// TIA Portal V15.1 export
// export: Created 2020-06-12T07:35:51.5537109Z, ExportSetting None, DisplayName Totally Integrated Automation Portal, DisplayVersion V15.1, DisplayName TIA Portal Openness, DisplayVersion V15.1, DisplayName STEP 7 Professional, DisplayVersion V15.1, DisplayName STEP 7 Safety, DisplayVersion V15.1, DisplayName WinCC Advanced, DisplayVersion V15.1
FUNCTION "MELT_Locks" : Void   // FC50, FBD
{ S7_Optimized_Access := 'TRUE' }
// stored: SetENOAutomatically False
   VAR_TEMP
      tCBisDisabled : Bool;
      tCBisLocked : Bool;
      tCWTripByMS : Bool;
      tCWPumpsStop : Bool;
      tMeltTripReset : Bool;
      tMpStatus : Word;
      tMeltTrip : Bool;
      tReset : Bool;
      tLC5MeltMode : Bool;
      tMSNotUsed : Bool;
   END_VAR
BEGIN

REGION Network 1: Reset trips
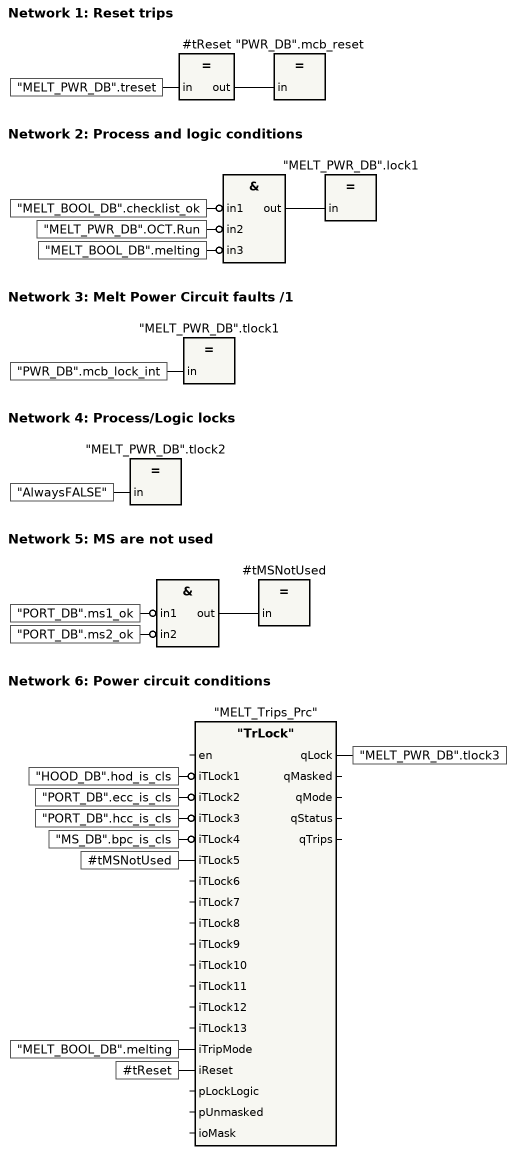
   #tReset := "MELT_PWR_DB".treset;
   "PWR_DB".mcb_reset := "MELT_PWR_DB".treset;
END_REGION

REGION Network 2: Process and logic conditions
   "MELT_PWR_DB".lock1 := NOT "MELT_BOOL_DB".checklist_ok AND NOT "MELT_PWR_DB".OCT.Run AND NOT "MELT_BOOL_DB".melting;
END_REGION

REGION Network 3: Melt Power Circuit faults /1
   "MELT_PWR_DB".tlock1 := "PWR_DB".mcb_lock_int;
END_REGION

REGION Network 4: Process/Logic locks
   // THIS IS TEMPORARY
   "MELT_PWR_DB".tlock2 := "AlwaysFALSE";
END_REGION

REGION Network 5: MS are not used
   #tMSNotUsed := NOT "PORT_DB".ms1_ok AND NOT "PORT_DB".ms2_ok;
END_REGION

REGION Network 6: Power circuit conditions
   "MELT_Trips_Prc"(iTLock1 := NOT "HOOD_DB".hod_is_cls,   // "TrLock"
                    iTLock2 := NOT "PORT_DB".ecc_is_cls,
                    iTLock3 := NOT "PORT_DB".hcc_is_cls,
                    iTLock4 := NOT "MS_DB".bpc_is_cls,
                    iTLock5 := #tMSNotUsed,
                    iTripMode := "MELT_BOOL_DB".melting,
                    iReset := #tReset,
                    qLock => "MELT_PWR_DB".tlock3);
END_REGION

REGION Network 7: Cooling common trips
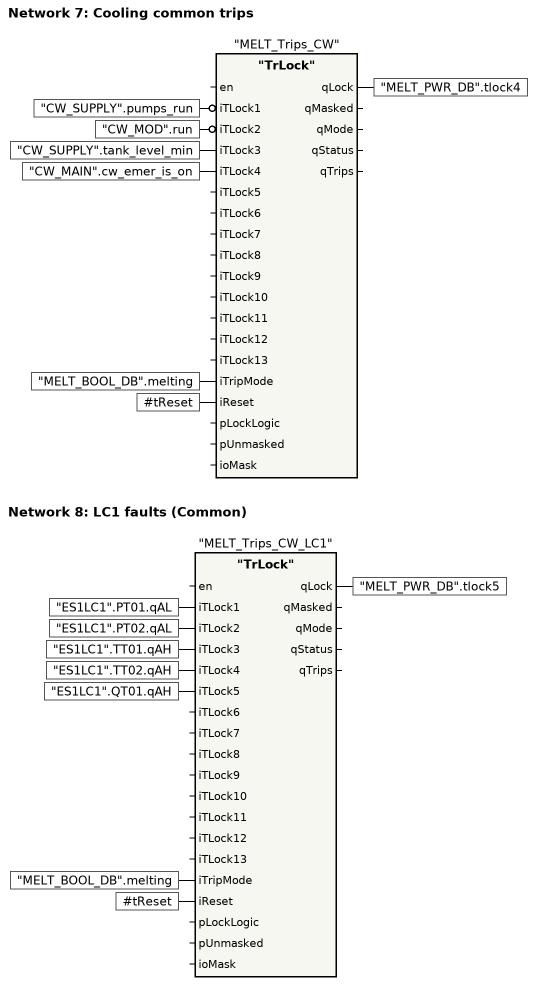
   "MELT_Trips_CW"(iTLock1 := NOT "CW_SUPPLY".pumps_run,   // "TrLock"
                   iTLock2 := NOT "CW_MOD".run,
                   iTLock3 := "CW_SUPPLY".tank_level_min,
                   iTLock4 := "CW_MAIN".cw_emer_is_on,
                   iTripMode := "MELT_BOOL_DB".melting,
                   iReset := #tReset,
                   qLock => "MELT_PWR_DB".tlock4);
END_REGION

REGION Network 8: LC1 faults (Common)
   // "ES1LC1".TT03.qAH
   // "ES1LC1".TT04.qAH
   "MELT_Trips_CW_LC1"(iTLock1 := "ES1LC1".PT01.qAL,   // "TrLock"
                       iTLock2 := "ES1LC1".PT02.qAL,
                       iTLock3 := "ES1LC1".TT01.qAH,
                       iTLock4 := "ES1LC1".TT02.qAH,
                       iTLock5 := "ES1LC1".QT01.qAH,
                       iTripMode := "MELT_BOOL_DB".melting,
                       iReset := #tReset,
                       qLock => "MELT_PWR_DB".tlock5);
END_REGION

REGION Network 9: LC3 faults (Portal + HC-clamps)
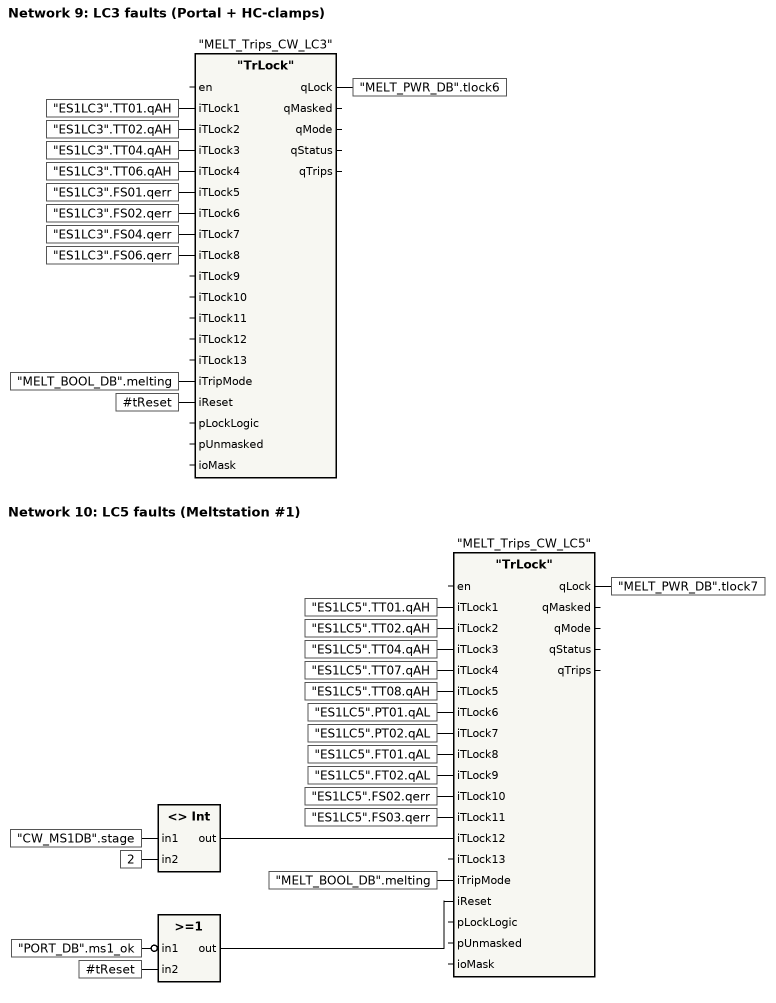
   "MELT_Trips_CW_LC3"(iTLock1 := "ES1LC3".TT01.qAH,   // "TrLock"
                       iTLock2 := "ES1LC3".TT02.qAH,
                       iTLock3 := "ES1LC3".TT04.qAH,
                       iTLock4 := "ES1LC3".TT06.qAH,
                       iTLock5 := "ES1LC3".FS01.qerr,
                       iTLock6 := "ES1LC3".FS02.qerr,
                       iTLock7 := "ES1LC3".FS04.qerr,
                       iTLock8 := "ES1LC3".FS06.qerr,
                       iTripMode := "MELT_BOOL_DB".melting,
                       iReset := #tReset,
                       qLock => "MELT_PWR_DB".tlock6);
END_REGION

REGION Network 10: LC5 faults (Meltstation #1)
   "MELT_Trips_CW_LC5"(iTLock1 := "ES1LC5".TT01.qAH,   // "TrLock"
                       iTLock2 := "ES1LC5".TT02.qAH,
                       iTLock3 := "ES1LC5".TT04.qAH,
                       iTLock4 := "ES1LC5".TT07.qAH,
                       iTLock5 := "ES1LC5".TT08.qAH,
                       iTLock6 := "ES1LC5".PT01.qAL,
                       iTLock7 := "ES1LC5".PT02.qAL,
                       iTLock8 := "ES1LC5".FT01.qAL,
                       iTLock9 := "ES1LC5".FT02.qAL,
                       iTLock10 := "ES1LC5".FS02.qerr,
                       iTLock11 := "ES1LC5".FS03.qerr,
                       iTLock12 := "CW_MS1DB".stage <> 2,
                       iTripMode := "MELT_BOOL_DB".melting,
                       iReset := NOT "PORT_DB".ms1_ok OR #tReset,
                       qLock => "MELT_PWR_DB".tlock7);
END_REGION

REGION Network 11: LC6 faults (Meltstation #2)
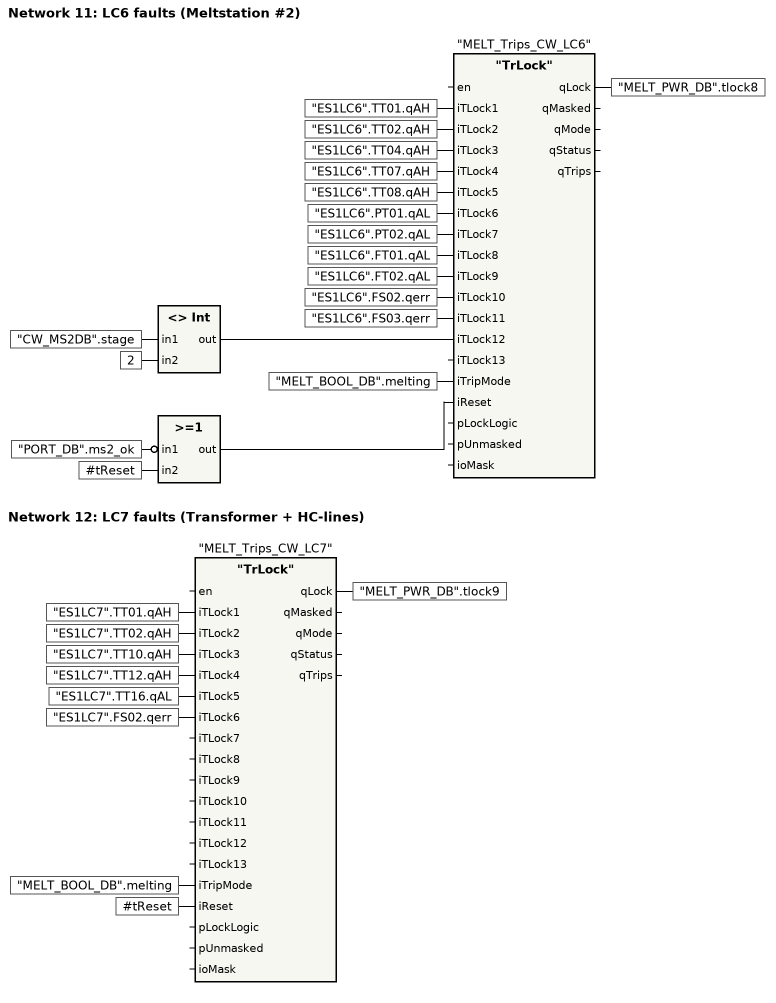
   "MELT_Trips_CW_LC6"(iTLock1 := "ES1LC6".TT01.qAH,   // "TrLock"
                       iTLock2 := "ES1LC6".TT02.qAH,
                       iTLock3 := "ES1LC6".TT04.qAH,
                       iTLock4 := "ES1LC6".TT07.qAH,
                       iTLock5 := "ES1LC6".TT08.qAH,
                       iTLock6 := "ES1LC6".PT01.qAL,
                       iTLock7 := "ES1LC6".PT02.qAL,
                       iTLock8 := "ES1LC6".FT01.qAL,
                       iTLock9 := "ES1LC6".FT02.qAL,
                       iTLock10 := "ES1LC6".FS02.qerr,
                       iTLock11 := "ES1LC6".FS03.qerr,
                       iTLock12 := "CW_MS2DB".stage <> 2,
                       iTripMode := "MELT_BOOL_DB".melting,
                       iReset := NOT "PORT_DB".ms2_ok OR #tReset,
                       qLock => "MELT_PWR_DB".tlock8);
END_REGION

REGION Network 12: LC7 faults (Transformer + HC-lines)
   // rlg 29/07/2019 
   // "ES1LC7".FS01.qerr
   // flow switch is not installed, flow transmiter is installed in the place
   "MELT_Trips_CW_LC7"(iTLock1 := "ES1LC7".TT01.qAH,   // "TrLock"
                       iTLock2 := "ES1LC7".TT02.qAH,
                       iTLock3 := "ES1LC7".TT10.qAH,
                       iTLock4 := "ES1LC7".TT12.qAH,
                       iTLock5 := "ES1LC7".TT16.qAL,
                       iTLock6 := "ES1LC7".FS02.qerr,
                       iTripMode := "MELT_BOOL_DB".melting,
                       iReset := #tReset,
                       qLock => "MELT_PWR_DB".tlock9);
END_REGION

REGION Network 13: Process trips
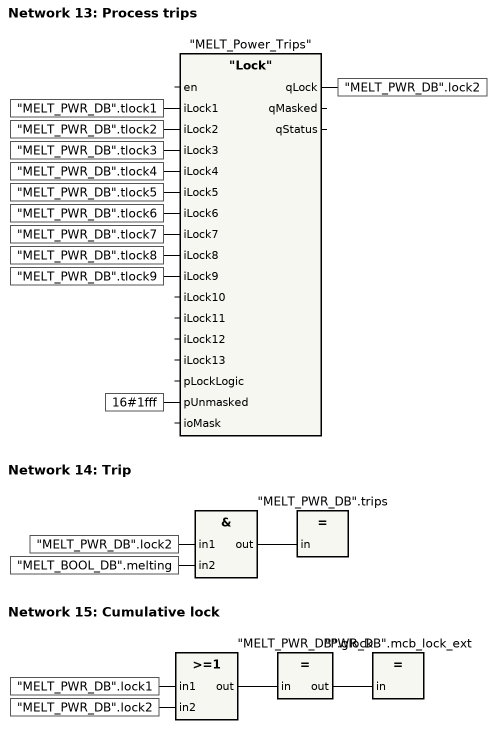
   "MELT_Power_Trips"(iLock1 := "MELT_PWR_DB".tlock1,   // "Lock"
                      iLock2 := "MELT_PWR_DB".tlock2,
                      iLock3 := "MELT_PWR_DB".tlock3,
                      iLock4 := "MELT_PWR_DB".tlock4,
                      iLock5 := "MELT_PWR_DB".tlock5,
                      iLock6 := "MELT_PWR_DB".tlock6,
                      iLock7 := "MELT_PWR_DB".tlock7,
                      iLock8 := "MELT_PWR_DB".tlock8,
                      iLock9 := "MELT_PWR_DB".tlock9,
                      pUnmasked := 16#1fff,
                      qLock => "MELT_PWR_DB".lock2);
END_REGION

REGION Network 14: Trip
   "MELT_PWR_DB".trips := "MELT_PWR_DB".lock2 AND "MELT_BOOL_DB".melting;
END_REGION

REGION Network 15: Cumulative lock
   "MELT_PWR_DB".glock := "MELT_PWR_DB".lock1 OR "MELT_PWR_DB".lock2;
   "PWR_DB".mcb_lock_ext := "MELT_PWR_DB".glock;
END_REGION

REGION Network 16: [[END]]
END_REGION
END_FUNCTION
